Yaskawa INFORM job: FRONT_WELD_90ST-1_4840.JBI

/JOB
//NAME FRONT_WELD_90ST-1_4840
///FOLDERNAME 02-SKRZYNIE_JOBS
//POS
///NPOS 31,31,0,6,0,0
///TOOL 0
///POSTYPE PULSE
///PULSE
C00000=0,-52278,40443,0,6873,1
C00001=0,-52278,40443,5610,-49281,72137
C00002=0,-42686,23640,7425,-34877,70985
C00003=25126,-44577,-4813,57071,-34461,49771
C00004=6017,-48449,-29001,102269,-8383,26407
C00005=2863,-32693,-8619,87056,-6043,33280
C00006=3232,-30428,-5975,86107,-6286,33771
C00007=3066,-30436,-5989,86105,-6179,33756
C00008=-22636,-29271,-6233,79447,10427,34222
C00009=-48870,-22313,-1449,76774,27638,32945
C00010=-50847,-28145,-10545,73666,29314,34422
C00011=-71330,-4959,8771,57572,20266,52624
C00012=-72821,-3113,10678,58516,21171,52061
C00013=-72538,1373,18723,63287,20013,49685
C00014=-72589,1362,18763,63564,20084,49594
C00015=-75601,1588,23023,78486,25219,45042
C00016=-69876,-3767,19948,87237,21294,41869
C00017=-54033,-13537,11070,98211,11134,38131
C00018=-58678,-17366,4552,88847,13968,42180
C00019=23545,-30165,-21390,32579,21562,60781
C00020=43411,-19640,-10965,-1347,18370,78573
C00021=44396,-17298,-7781,-3280,17967,79574
C00022=44355,-17319,-7798,-3202,17962,79534
C00023=50167,-19817,-7183,-40985,20083,89431
C00024=52866,-20120,-9469,-47174,28956,86193
C00025=41936,-24575,-13047,-39192,23123,81393
C00026=22415,-29011,-20931,-6356,22431,64332
C00027=24971,-35737,-30976,-9397,24510,66000
C00028=0,-42686,23640,7425,-34877,70985
C00029=0,-52278,40443,5610,-49281,72137
C00030=0,-52278,40443,0,6873,1
BC00000=744037
BC00001=744037
BC00002=872318
BC00003=909953
BC00004=940778
BC00005=940778
BC00006=940779
BC00007=940779
BC00008=940780
BC00009=940779
BC00010=940779
BC00011=940780
BC00012=940780
BC00013=940780
BC00014=940780
BC00015=940780
BC00016=940840
BC00017=940780
BC00018=940780
BC00019=940780
BC00020=940779
BC00021=940779
BC00022=940779
BC00023=940779
BC00024=940779
BC00025=940779
BC00026=940779
BC00027=940779
BC00028=872318
BC00029=744037
BC00030=744037
///POSTYPE BASE
///RECTAN
///RCONF 1,0,0,0,0,0,0,0,0,0,0,0,0,0,0,0,0,0,0,0,0,0,0,0
P00500=2.332,-5.281,-1.258,0.0000,0.0000,0.0000
///RCONF 0,0,0,0,0,0,0,0,0,0,0,0,0,0,0,0,0,0,0,0,0,0,0,0
P00501=-2.026,0.009,3.534,0.0000,0.0000,0.0000
///RCONF 1,0,0,0,0,0,0,0,0,0,0,0,0,0,0,0,0,0,0,0,0,0,0,0
P00502=-2.023,0.001,1.732,0.0000,0.0000,0.0000
P00503=0.138,-0.044,1.539,0.0000,0.0000,0.0000
P00504=-0.309,-0.010,1.636,0.0000,0.0000,0.0000
P00505=0.999,-9.916,8.214,0.0000,0.0000,0.0000
//INST
///DATE 2024/07/03 16:33
///ATTR SC,RW
///GROUP1 RB1,BS1
NOP
MOVJ C00000 BC00000 VJ=50.00
MOVJ C00001 BC00001 VJ=50.00
MOVJ C00002 BC00002 VJ=50.00
MOVJ C00003 BC00003 VJ=50.00
MOVJ C00004 BC00004 VJ=30.00
'::::::::::::::::::::::::::::::::
'W20
'::::::::::::::::::::::::::::::::
MOVL C00005 BC00005 V=333.3
SFTON P0503
MACRO1 MJ#(0) ARGF14
MOVL C00006 BC00006 V=133.3 PL=0
ARCON
MOVC C00007 BC00007 V=9.5
MOVC C00008 BC00008 V=9.5
SFTOF
SFTON P0502
MOVC C00009 BC00009 V=9.5
ARCOF
MOVL C00010 BC00010 V=250.0
SFTOF
MOVL C00011 BC00011 V=250.0
'::::::::::::::::::::::::::::::::
'W21
'::::::::::::::::::::::::::::::::
MOVL C00012 BC00012 V=166.7
SFTON P0500
MACRO1 MJ#(0) ARGF14
MOVL C00013 BC00013 V=133.3 PL=0
ARCON
MOVC C00014 BC00014 V=9.5
MOVC C00015 BC00015 V=9.5
MOVC C00016 BC00016 V=9.5
SFTOF
SFTON P0501
MOVC C00017 BC00017 V=9.5
ARCOF
MOVL C00018 BC00018 V=250.0
SFTOF
MOVL C00019 BC00019 V=333.3
'::::::::::::::::::::::::::::::::
'W22
'::::::::::::::::::::::::::::::::
MOVL C00020 BC00020 V=166.7
SFTON P0505
MACRO1 MJ#(0) ARGF14
MOVL C00021 BC00021 V=133.3 PL=0
ARCON
MOVC C00022 BC00022 V=9.5
MOVC C00023 BC00023 V=9.5
MOVC C00024 BC00024 V=9.5
SFTOF
SFTON P0504
MOVC C00025 BC00025 V=9.5
MOVC C00026 BC00026 V=9.5
ARCOF
MOVL C00027 BC00027 V=166.7
SFTOF
MOVJ C00028 BC00028 VJ=50.00
MOVJ C00029 BC00029 VJ=80.00
MOVJ C00030 BC00030 VJ=80.00
END
